Staubli VAL3: statistics.pjx

--- statistics.pjx ---
Parameters version=s8.12Cs9_BS2378 stackSize=5000 millimeterUnit=true
Program file=getGeometricMean.pgx
Program file=getHarmonicMean.pgx
Program file=getMean.pgx
Program file=getMedian.pgx
Program file=getStandardDeviation.pgx
Program file=getVariance.pgx
Program file=start.pgx
Program file=stop.pgx
Data file=statistics.dtx

--- statistics.dtx ---
mdesc mNomSpeed
num nTemp
num nInput[8]
num nCopy

--- start.pgx ---
program start()
  local num l_nMean
  local num l_nMedian
  local num l_nVariance
  local num l_nStandardDeviation
  local num l_nGeoMean
  local num l_nRes
begin

  nInput[0] = 2
  nInput[1] = 1
  nInput[2] = 6
  nInput[3] = 5
  nInput[4] = 2
  nInput[5] = 4
  nInput[6] = 1
  nInput[7] = 7

  call getMean(nInput, l_nRes)
  ? "Mittelwert: " + toString(".4", l_nRes)

  call getMedian(nInput, l_nRes)
  ? "Median: " + toString(".4", l_nRes)

  call getVariance(nInput, l_nRes)
  ? "Varianz: " + toString(".4", l_nRes)

  call getStandardDeviation(nInput, l_nRes)
  ? "Std. Deviation: " + toString(".4", l_nRes)

  call getGeometricMean(nInput, l_nRes)
  ? "Geom. Mean: " + toString(".4", l_nRes)

  call getHarmonicMean(nInput, l_nRes)
  ? "Harm. Mean: " + toString(".4", l_nRes)
end

--- getGeometricMean.pgx ---
public program getGeometricMean(num& x_nInput[], num& x_nMean)
  local num l_nCount
  local num l_nProd
begin

  l_nProd = 1

  for l_nCount = 0 to size(x_nInput)-1
    l_nProd = l_nProd * x_nInput[l_nCount]
  endFor
  ? l_nProd
  x_nMean = power(l_nProd,1/size(x_nInput))

end

--- getHarmonicMean.pgx ---
public program getHarmonicMean(num& x_nInput[], num& x_nMean)
  local num l_nCount
  local num l_nSum
begin

  l_nSum = 0

  for l_nCount = 0 to size(x_nInput)-1
    l_nSum = l_nSum + 1/x_nInput[l_nCount]
  endFor

  x_nMean = size(x_nInput)/ l_nSum

end

--- getMean.pgx ---
public program getMean(num& x_nInput[], num& x_nMean)
  local num l_nCount
  local num l_nSum
begin

  l_nSum = 0

  for l_nCount = 0 to size(x_nInput)-1
    l_nSum = l_nSum + x_nInput[l_nCount]
  endFor

  x_nMean = l_nSum/size(x_nInput)

end

--- getMedian.pgx ---
public program getMedian(num& x_nInput[], num& x_nMedian)
  local num l_nCount
  local num l_nSmallsub
  local num l_nSort
  local num l_nTemp
begin

  // do a selection sort:
  // The idea of Selection Sort is that we repeatedly find the smallest element in the unsorted part of the array and swap it with the first element in the unsorted part of the array.

  resize(nTemp, 1, size(x_nInput))
  resize(nCopy, 1, size(x_nInput))

  for l_nCount = 0 to size(x_nInput)-1
    nCopy[l_nCount] = x_nInput[l_nCount]
  endFor


  for l_nCount = 0 to size(nCopy)-1
    l_nSmallsub = l_nCount

    for l_nSort = l_nCount+1 to size(nCopy)-1
      if nCopy[l_nSort] < nCopy[l_nSmallsub]
        l_nSmallsub = l_nSort
      endIf
    endFor

    l_nTemp = nCopy[l_nCount]
    nTemp[l_nCount] = nCopy[l_nSmallsub]
    nCopy[l_nSmallsub] = l_nTemp

  endFor

  if size(nCopy)%2 != 0
    // extract middle value of sorted list
    x_nMedian = nTemp[((size(nCopy)+1)/2)-1]
  else
    x_nMedian = (nTemp[(size(nCopy)/2)-1] + nTemp[size(nCopy)/2])/2
  endIf


end

--- getStandardDeviation.pgx ---
public program getStandardDeviation(num& x_nInput[], num& x_nStandardDeviation)
  local num l_nVariance
begin

  call getVariance(x_nInput, l_nVariance)

  x_nStandardDeviation = sqrt(l_nVariance)
end

--- getVariance.pgx ---
public program getVariance(num& x_nInput[], num& x_nVariance)
  local num l_nMean
  local num l_nCount
  local num l_nSum
begin

  l_nSum = 0
  // get mean of the input numbers
  call getMean(x_nInput, l_nMean)

  for l_nCount = 0 to size(x_nInput)-1
    l_nSum = l_nSum + power(x_nInput[l_nCount]-l_nMean, 2)
  endFor

  x_nVariance = l_nSum/size(x_nInput)

end
